FUNCTION_BLOCK FB_StateMachine
VAR_INPUT
    stFaults    		: ST_Faults;
    stHmiSetpoints 		: ST_HmiSetpoints;
	stProcessValues		: ST_ProcessValues;
	bDeliveryCmd		: BOOL;
	bFillComplete		: BOOL;
	bPurgeComplete		: BOOL;
	rSpaTemp			: REAL;
	bSpaFlushed			: BOOL;
END_VAR
VAR_OUTPUT
	// system state
    eState           : E_SystemState := E_SystemState.InitController;
    // enable flags for downstream FBs
	eWaterFillMode 	 : E_WaterFillMode;   	// water fill mode startup/autofill/idle
	bControlEnable   : BOOL;   				// PID pressure/temp loops may run
    bPurgeEnable     : BOOL;   				// vessel purge sequence active
	bSpaFlushEnable	 : BOOL;				// enable SPA flush sequence
	bSpaFlushReset	 : BOOL;				// reset SPA flush fb
	bDeliveryEnable	 : BOOL;				// enable steam delivery
    bReady           : BOOL;   				// green Ready: in SteamFlowing, in-band, no faults
    bInStartup       : BOOL;   				// TRUE for any Init* state
END_VAR
VAR
    // --- request flags set by methods, cleared when serviced ---
    bReqStart        : BOOL;
    bReqStop         : BOOL;
    bReqMaint        : BOOL;
    bReqExitMaint    : BOOL;
    bReqFault        : BOOL;
    bReqFaultReset   : BOOL;
    // --- state entry detection (rising edge of a new state) ---
    eStatePrev       : E_SystemState;
    bEntry           : BOOL;   // TRUE on the first cycle of the current state
	// TODO move to fbFaultMonitor and delete from here
    // --- thresholds (seed from GVL_Params at init; defaults from source) ---
    tWarmupTime      : TIME := T#120S;   // legacy "Begin a 120 sec warm up timer for TC3"
    tDiffPressTime   : TIME := T#10M;    // legacy baseline 15 min
    tFillTimeout     : TIME := T#10M;
    tPurgeTimeout    : TIME := T#10M;
END_VAR

//=========================== entry-edge detection ============================
bEntry := (eState <> eStatePrev);
eStatePrev := eState;

//=========================== reset on entry detection ========================
IF bEntry THEN	
	// do something
END_IF

//=========================== global fault override ===========================
// A latching fault forces Fault from ANY state except when already resetting.
IF bReqFault AND (eState <> E_SystemState.Fault) THEN
    eState := E_SystemState.Fault;
    bEntry := TRUE;
END_IF
bReqFault := FALSE;

//=========================== default enable flags ============================
// Recomputed every cycle; each state turns on what it needs below.
eWaterFillMode 	:= E_WaterFillMode.Idle;
bControlEnable  := FALSE;
bPurgeEnable    := FALSE;
bSpaFlushEnable := FALSE;
bSpaFlushReset  := FALSE;
bDeliveryEnable := FALSE;
bReady          := FALSE;
bInStartup      := FALSE;

//================================ STATE MACHINE ==============================
CASE eState OF

    //--------------------------------------------------------------------
    E_SystemState.InitController:   // S0 : one-shot init, then idle
    //--------------------------------------------------------------------
        IF bEntry THEN
            // TODO: seed thresholds from GVL_Params here if they differ per unit
            ;
        END_IF
        eState := E_SystemState.SesOff;

    //--------------------------------------------------------------------
    E_SystemState.SesOff:           // S70 : SES off, idle / standby
    //--------------------------------------------------------------------
        IF bReqMaint THEN
            eState := E_SystemState.Maintenance;
        ELSIF stFaults.bAnyFault THEN
			bReqFault := TRUE;
		ELSIF bReqStart AND NOT stFaults.bHmiCommLoss THEN
            eState := E_SystemState.CheckIfHot;
        END_IF

    //--------------------------------------------------------------------
    E_SystemState.CheckIfHot:       // S10 : hot-restart shortcut vs cold start
    //--------------------------------------------------------------------
        // SPA warm (TC1 within band) AND steam flow already > x%*RatedFlow -> jump to SteamFlowing.
        // Otherwise cold start -> fill water
        bInStartup := TRUE;
        IF _IsSpaWarm() AND (_FlowPercent() > GVL_SysParameters.rHotRestartFlowPct) THEN
            eState := E_SystemState.SteamFlowing;
		ELSE
            eState := E_SystemState.FillWater;
        END_IF

    //--------------------------------------------------------------------
    E_SystemState.FillWater:    // S20 : fill water
    //--------------------------------------------------------------------
        bInStartup      := TRUE;
        eWaterFillMode 	:= E_WaterFillMode.StartupFill;

        IF bReqStop THEN
            eState := E_SystemState.SesOff;
        ELSIF stFaults.bAnyFault THEN
            bReqFault := TRUE;  
        ELSIF bFillComplete THEN
			IF GVL_HMI.stHmiSetpoints.bSetPurgeOnStartup THEN 
				eState := E_SystemState.PurgeVessel;
			ELSE 
				eState := E_SystemState.SetDiffPressure; 
			END_IF
        END_IF

    //--------------------------------------------------------------------
    E_SystemState.PurgeVessel:  // S30 : purge vessel
    //--------------------------------------------------------------------
        bInStartup   := TRUE;
        bPurgeEnable := TRUE;
		bControlEnable := TRUE;

		// Blowdown first, refill second
		IF bPurgeComplete THEN
			eWaterFillMode := E_WaterFillMode.StartupFill;   // legacy rung 114
		ELSE
			eWaterFillMode := E_WaterFillMode.Idle;          // legacy rung 103: "do not fill water until purge complete"
		END_IF

        IF bReqStop THEN
            eState := E_SystemState.SesOff;
        ELSIF stFaults.bAnyFault THEN
            bReqFault := TRUE;
        ELSIF bPurgeComplete AND bFillComplete THEN
            eState := E_SystemState.SetDiffPressure;
        END_IF

    //--------------------------------------------------------------------
    E_SystemState.SetDiffPressure: // S40 : establish differential pressure
    //--------------------------------------------------------------------
        bInStartup     := TRUE;
        bControlEnable := TRUE;   // dP PID runs to bring differential up

        IF bReqStop THEN
            eState := E_SystemState.SesOff;
		ELSIF stFaults.bAnyFault THEN
            bReqFault := TRUE;    // legacy DS start-high -> S10
        ELSIF _DiffPressEstablished() THEN
            eState := E_SystemState.InitMain;
        END_IF

    //--------------------------------------------------------------------
    E_SystemState.InitMain:         // S50 : final checks before flow
    //--------------------------------------------------------------------
    bInStartup     := TRUE;
    bControlEnable := TRUE;
    bSpaFlushEnable := TRUE;
    eWaterFillMode := E_WaterFillMode.RunningAutofill;

    IF bReqStop THEN
        eState := E_SystemState.SesOff;
	ELSIF stFaults.bAnyFault THEN
		bReqFault := TRUE;
    ELSIF bSpaFlushed AND _TempsInBand() AND _FlowInBand() THEN
        eState := E_SystemState.SteamFlowing;
    END_IF

    //--------------------------------------------------------------------
    E_SystemState.SteamFlowing:     // S60: normal production
    //--------------------------------------------------------------------
        bControlEnable := TRUE;
		eWaterFillMode := E_WaterFillMode.RunningAutofill;
        // Ready = producing, no active faults, flow tracking setpoint
        bReady := NOT stFaults.bAnyFault
                  AND _FlowInBand()
                  AND _TempsInBand();
		
		bDeliveryEnable := bDeliveryCmd AND NOT stFaults.bHmiCommLoss;
				  
        IF bReqStop THEN
            eState := E_SystemState.SesOff;
		ELSIF stFaults.bAnyFault THEN
			bReqFault := TRUE;
        END_IF

    //--------------------------------------------------------------------
    E_SystemState.Maintenance:      // S80 : manual actuation
    //--------------------------------------------------------------------
        // Outputs handled by FB_OutputHandler via HMI overrides; no auto control.
		bControlEnable := NOT stFaults.bHmiCommLoss;
		
		IF bReqExitMaint OR bReqStop THEN
			eState := E_SystemState.SesOff;
		ELSIF stFaults.bAnyFault THEN
			bReqFault := TRUE;
		END_IF

    //--------------------------------------------------------------------
    E_SystemState.Fault:            // S99 : latched fault
    //--------------------------------------------------------------------
        // All auto outputs off. Only an operator reset leaves this state,
        // and only once all latching faults have actually cleared.
        // Operator reset: clear latches, then let the monitor re-evaluate.

		IF bReqFaultReset AND NOT stFaults.bHmiCommLoss THEN
            eState := E_SystemState.InitController;
        END_IF

ELSE
    // Unknown/illegal state -> safe fallback
    eState := E_SystemState.Fault;
END_CASE

//=========================== clear serviced requests =========================
// (bReqFault is cleared at the top of the next cycle after being serviced.)
bReqStart      := FALSE;
bReqStop       := FALSE;
bReqMaint      := FALSE;
bReqExitMaint  := FALSE;
bReqFaultReset := FALSE;

// TODO: real dP target from setpoints/params (legacy "Purge dP"/INI_SP).
METHOD PRIVATE _DiffPressEstablished : BOOL
_DiffPressEstablished := (stProcessValues.rDiffPressure >= stHmiSetpoints.rSetDsPressure);
END_METHOD

METHOD PRIVATE _FlowInBand : BOOL
// check if measured flow is within tolerance of setpoint for hot start
_FlowInBand := ABS(stProcessValues.rFlowActual - stHmiSetpoints.rSetFlow) <= (GVL_SysParameters.rFlowDeadbandPct * stHmiSetpoints.rSetFlow);
END_METHOD

METHOD PRIVATE _FlowPercent : REAL
IF stProcessValues.rFlowRated > 0.0 THEN
    _FlowPercent := 100.0 * stProcessValues.rFlowActual / stProcessValues.rFlowRated;
ELSE
    _FlowPercent := 0.0;
END_IF
END_METHOD

METHOD PRIVATE _IsSpaWarm : BOOL
_IsSpaWarm := (stProcessValues.rTc1Spa >= GVL_SysParameters.rSpaWarmMinimumTemp);
END_METHOD

// TODO: real temperature bands from params (Warmup Temp V1535, Max Temp V1522).
METHOD PRIVATE _TempsInBand : BOOL
_TempsInBand := (rSpaTemp >= 30.0) AND (rSpaTemp <= 130.0);
END_METHOD

METHOD RequestExitMaint : BOOL
bReqExitMaint := TRUE;
RequestExitMaint := TRUE;
END_METHOD

// Force Fault. Called by MAIN when FB_FaultMonitor latches a fault.
METHOD RequestFault : BOOL
bReqFault := TRUE;
RequestFault := TRUE;
END_METHOD

// Operator reset. Only leaves Fault when latching faults have cleared.
METHOD RequestFaultReset : BOOL
bReqFaultReset := TRUE;
RequestFaultReset := TRUE;
END_METHOD

// Enter Maintenance. Honored only from SesOff.
METHOD RequestMaintenance : BOOL
bReqMaint := TRUE;
RequestMaintenance := TRUE;
END_METHOD

// SES ON. Honored only from SesOff (checked in the CASE).
METHOD RequestStart : BOOL
bReqStart := TRUE;
RequestStart := TRUE;
END_METHOD

// SES OFF / abort. Honored from any running or startup state.
METHOD RequestStop : BOOL
bReqStop := TRUE;
RequestStop := TRUE;
END_METHOD

END_FUNCTION_BLOCK

(* stored: Version 1.1.0.1, ProductVersion 3.1.4026.18
   POU FB_StateMachine: Id {c229f4cc-9a87-4d59-a1ae-d17bbe58764f}, SpecialFunc None
   Method _DiffPressEstablished: Id {b1f7aed4-a886-4a7b-bad9-cc81f3fbcb42}
   Method _FlowInBand: Id {7b34b003-618c-4463-9a96-27a32ac34e28}
   Method _FlowPercent: Id {51f9c619-5222-4c48-a32b-707ad7ce6221}
   Method _IsSpaWarm: Id {79115b31-84d2-410e-8a34-0a55ab06bbbe}
   Method _TempsInBand: Id {d3fe4c13-f97f-4432-8bcd-b18afa8468b0}
   Method RequestExitMaint: Id {d6350887-01b9-4198-9246-356e4bc00618}
   Method RequestFault: Id {a61af9d8-4978-47f2-84b4-896606f3e70c}
   Method RequestFaultReset: Id {87dbab1b-7fca-4407-aed1-430ea9e709b2}
   Method RequestMaintenance: Id {44772f76-bcc8-4a70-8395-cccc8d10bb8d}
   Method RequestStart: Id {bac3a0e4-aadf-4d2f-b000-40664aac8f98}
   Method RequestStop: Id {1d1b5f77-76a5-45dc-a6eb-c9f10c103138} *)
